(* launch IE browser window to browse MV420/MV440 at specified IP address *)
FUNCTION_BLOCK FB_CAMERA_OmronBrowse
VAR_INPUT
	bViewLive		: BOOL;		(* set TRUE to view live images from MV4x0 scanner *)
	bViewDiag		: BOOL;		(* set TRUE to view failed images from MV4x0 scanner *)
	sIPAddress		: T_IPv4Addr;	(* IP address of scanner *)
END_VAR
VAR_OUTPUT
	bDone			: BOOL;		(* TRUE = launch browser complete *)
	bBusy			: BOOL;		(* TRUE = launch browser in progress *)
	bError			: BOOL;		(* TRUE = error when launching browser *)
	nErrorID		: UDINT;	(* error code *)
END_VAR
VAR
	bExecute		: BOOL;
	fbExecute		: R_TRIG;
	eState			: E_CAMERA_State;
	fbCheckOS		: FB_CAMERA_CheckOS;
	sDirectory		: STRING(39);
	sBrowser		: STRING(15);
	sCommandParam	: STRING(255);
	fbStartProcess	: NT_StartProcess;
END_VAR

(* browse scanner on rising edge of bViewLive or bViewDiag *)
bExecute := bViewLive = TRUE OR bViewDiag = TRUE;
fbExecute(CLK := bExecute);

CASE eState OF

	(* IDLE state *)
	E_CAMERA_State.IDLE:

		(* rising edge of bExecute *)
		IF fbExecute.Q = TRUE THEN

			(* update outputs *)
			bDone := FALSE;
			bBusy := TRUE;
			bError := FALSE;
			nErrorID := 0;

			(* view live images from scanner *)
			IF bViewLive = TRUE THEN

				(* address for live image view *)
(*				strCommandParam := F_CONCAT3('http://', strIPAddress, '/peeklive.html');*)
				sCommandParam := CONCAT('http://', sIPAddress);

			(* view diagnostic images from scanner *)
			ELSIF bViewDiag = TRUE THEN

				(* address for diagnostic image view *)
(*				strCommandParam := F_CONCAT3('http://', strIPAddress, '/ediagimghtml.cgi'); *)
				sCommandParam := CONCAT('http://', sIPAddress);
			END_IF

			eState := E_CAMERA_State.CHECKOS;

		(* bExecute has been reset *)
		ELSIF bExecute = FALSE THEN

			(* reset outputs *)
			bDone := FALSE;
			bBusy := FALSE;
			bError := FALSE;
			nErrorID := 0;
		END_IF


	(* check local operating system *)
	E_CAMERA_State.CHECKOS:

		(* check OS  *)
		fbCheckOS(bExecute := TRUE);

		(* check OS complete *)
		IF fbCheckOS.bDone = TRUE THEN

			(* check OS completed OK *)
			IF fbCheckOS.bError = FALSE THEN

				(* OS is WinCE *)
				IF fbCheckOS.eOSType = E_OS_WINCE THEN

					sDirectory := '\Windows';
					sBrowser := '\iesample.exe';

				(* not WinCE, assume WinXP or similar *)
				ELSE

					sDirectory := 'C:\Program Files\Internet Explorer';
					sBrowser := '\iexplore.exe';
				END_IF

				eState := E_CAMERA_State.BROWSEDIAG;

			(* check OS error *)
			ELSE

				bError := FALSE;
				nErrorID := fbCheckOS.nErrorID;

				eState := E_CAMERA_State.DONE;
			END_IF

			(* clsoe off fbCheckOS *)
			fbCheckOS(bExecute := FALSE);
		END_IF


	(* start Internet Explorer *)
	E_CAMERA_State.BROWSEDIAG:

		(* start process *)
		fbStartProcess(
			NETID		:= '',
			PATHSTR		:= CONCAT(sDirectory, sBrowser),
			DIRNAME		:= sDirectory,
			COMNDLINE	:= sCommandParam,
			START		:= TRUE,
		);

		(* start process complete *)
		IF fbStartProcess.BUSY = FALSE THEN

			(* start process error *)
			IF fbStartProcess.ERR = TRUE THEN

				bError := TRUE;
				nErrorID := fbStartProcess.ERRID;
			END_IF

			eState := E_CAMERA_State.DONE;

			(* close off fbStartProcess *)
			fbStartProcess(START := FALSE);
		END_IF


	(* DONE state *)
	E_CAMERA_State.DONE:

		bBusy := FALSE;
		bDone := TRUE;

		eState := E_CAMERA_State.IDLE;


(* unknown state *)
ELSE

	eState := E_CAMERA_State.IDLE;
END_CASE

END_FUNCTION_BLOCK

(* stored: Version 1.1.0.1
   POU FB_CAMERA_OmronBrowse: Id {23ca150a-c0af-426c-9cd9-547f845927c6}, SpecialFunc None *)
